Staubli VAL3: TrajectoryItem.pjx

--- TrajectoryItem.pjx ---
Parameters version=s7.2.1 stackSize=5000 millimeterUnit=true
Data file=TrajectoryItem.dtx
Type name=InstrItem path=Disk://kernel/template/InstrItem/InstrItem.pjx

--- TrajectoryItem.dtx ---
public num distance
public num moveType
public num nTime
public num nStop
public num nTcpAction
public string comment
public bool toStop
public mdesc nom_speed = {vel=450, tmax=1000}
public InstrItem iInstr[3]
  [0]
    string sType
    string sData
  [1]
    string sType
    string sData
  [2]
    string sType
    string sData
public num nMoveId
